PROGRAM MAIN
VAR
	i: INT;
	
	Int2: INT;
END_VAR

i:=i+1;
Int2 :=Int2+1;

END_PROGRAM

(* stored: Version 1.1.0.1
   POU MAIN: Id {9874e98c-7aae-49e9-8032-680c1af470cf}, SpecialFunc None *)
